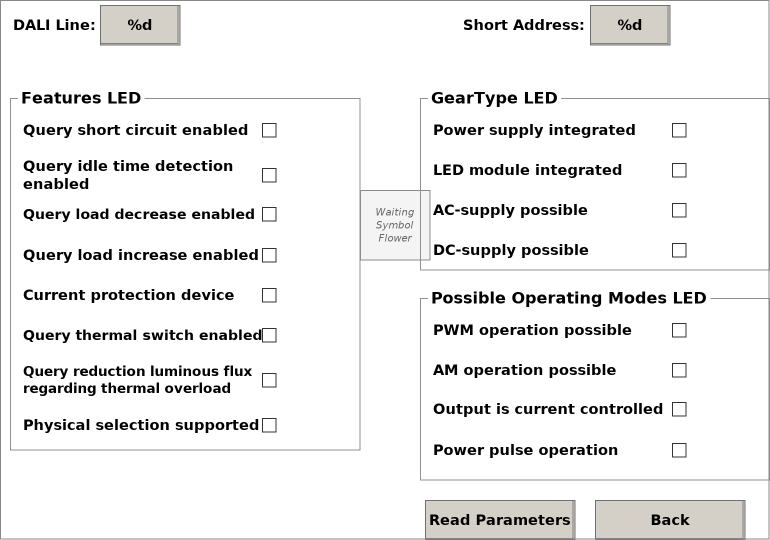
VISUALIZATION Visu_Part207Parameters  // 770x540
    Button (425,500 150x40), "Read Parameters"
        OnMouseClick: execute { DALI_Commissioning.fbPart207ParametersLED.bRead:=TRUE; }
    WaitingSymbolFlower (360,190 70x70), invisible if: DALI_Commissioning.fbPart207ParametersLED.bHideWaitSymbol
    GroupBox (420,90 350x180), "GearType LED"
        Textfield (10,25 220x30), "Power supply integrated"
        Checkbox (250,25 30x30), variable: DALI_Commissioning.fbPart207ParametersLED.bLEDPowerSupply
        Textfield (10,65 170x30)
        Textfield (10,65 220x30), "LED module integrated"
        Textfield (10,145 220x30), "DC-supply possible"
        Textfield (10,105 220x30), "AC-supply possible"
        Checkbox (250,65 30x30), variable: DALI_Commissioning.fbPart207ParametersLED.bLEDModule
        Checkbox (250,145 30x30), variable: DALI_Commissioning.fbPart207ParametersLED.bDCSupply
        Checkbox (250,105 30x30), variable: DALI_Commissioning.fbPart207ParametersLED.bACSupply
    GroupBox (10,90 350x360), "Features LED"
        Textfield (10,25 240x30), "Query short circuit enabled"
        Checkbox (250,25 30x30), variable: DALI_Commissioning.fbPart207ParametersLED.bQueryShortCircuitEnabled
        Textfield (10,65 240x30)
        Textfield (10,65 240x40), "Query idle time detection enabled"
        Textfield (10,150 240x30), "Query load increase enabled"
        Textfield (10,109 240x30), "Query load decrease enabled"
        Checkbox (250,70 30x30), variable: DALI_Commissioning.fbPart207ParametersLED.bQueryIdleTimeDetectionEnabled
        Checkbox (250,150 30x30), variable: DALI_Commissioning.fbPart207ParametersLED.bQueryLoadIncreaseEnabled
        Checkbox (250,109 30x30), variable: DALI_Commissioning.fbPart207ParametersLED.bQueryLoadDecreaseEnabled
        Textfield (10,190 240x30), "Current protection device"
        Checkbox (250,190 30x30), variable: DALI_Commissioning.fbPart207ParametersLED.bQueryCurrentProtectionDevicePresent
        Checkbox (250,230 30x30), variable: DALI_Commissioning.fbPart207ParametersLED.bQueryThermalSwitchEnabled
        Checkbox (250,275 30x30), variable: DALI_Commissioning.fbPart207ParametersLED.bQueryReductionOfLuminouFluxRegardingThermalOverloadEnabled
        Checkbox (250,320 30x30), variable: DALI_Commissioning.fbPart207ParametersLED.bPhysicalSelectionSupported
        Textfield (10,230 240x30), "Query thermal switch enabled"
        Textfield (10,270 240x40), "Query reduction luminous flux regarding thermal overload"
        Textfield (10,320 240x30), "Physical selection supported"
    Button (595,500 150x40), "Back"
        OnMouseClick: change screen: Previous 
    Group (460,5 210x40)
        Textfield (0,0 130x40), "Short Address:"
        Button (130,0 80x40), "%d", text variable: DALI_Commissioning.fbPart207ParametersLED.nAddress
            OnMouseClick: write the text variable via Default, min 0, max 63, title "Insert Short Address"
    Group (10,5 170x40)
        Textfield (0,0 110x40), "DALI Line:"
        Button (90,0 80x40), "%d", text variable: GVL_Internal.nDALILine
            OnMouseClick: write the text variable via Default, min 1, max 10, title "Choose line"
    GroupBox (420,290 350x190), "Possible Operating Modes LED", invisible if: DALI_Commissioning.fbPart207ParametersLED.bInvisible
        Checkbox (250,25 30x30), variable: DALI_Commissioning.fbPart207ParametersLED.bPWMOperation
        Textfield (10,65 240x30)
        Textfield (10,65 240x30), "AM operation possible"
        Textfield (10,145 240x30), "Power pulse operation"
        Textfield (10,104 240x30), "Output is current controlled"
        Checkbox (250,65 30x30), variable: DALI_Commissioning.fbPart207ParametersLED.bAMOperation
        Checkbox (250,145 30x30), variable: DALI_Commissioning.fbPart207ParametersLED.bPowerPulseOperation
        Checkbox (250,104 30x30), variable: DALI_Commissioning.fbPart207ParametersLED.bOutputCurrentControlled
        Textfield (10,25 240x30), "PWM operation possible"
END_VISUALIZATION

(* stored: Version 1.1.0.1, ProductVersion 3.1.4024.9
   Visu Visu_Part207Parameters: Id {4da47d3e-8855-4f6c-a557-60855b37564a} *)
